ABB RAPID module: RsTempModule.mod

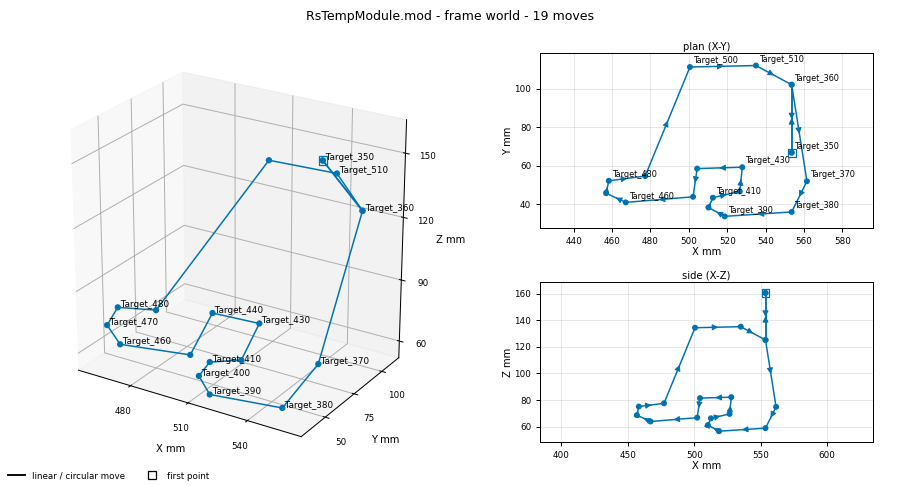
[picture p0: tool path of RsTempModule.mod in frame world, 19 of 19 moves have a stored position in this frame; points joined in program order, loops and branches not executed]
MODULE RsTempModule
    LOCAL CONST robtarget Target_350:=[[-145.225874554,122.068654602,-50.082052893],[0.707106781,0.000000819,-0.000000819,-0.707106781],[1,1,0,7],[9E+09,9E+09,9E+09,9E+09,9E+09,9E+09]];
    LOCAL PERS tooldata Portamarcador:=[TRUE,[[105.653,-1.591,36.465],[0.707106781,0,0.707106781,0]],[0.25,[0,0,1],[1,0,0,0],0,0,0]];
    LOCAL PERS wobjdata Tablero:=[FALSE,TRUE,"",[[0,0,0],[1,0,0,0]],[[431.492,204.933,227.769],[0.270598807,-0.653281169,-0.653281169,-0.270598807]]];
    LOCAL CONST robtarget Target_360:=[[-145.225990414,122.068654602,-0.082052893],[0.707106781,0.000000819,-0.000000819,-0.707106781],[0,0,0,1],[9E+09,9E+09,9E+09,9E+09,9E+09,9E+09]];
    LOCAL CONST robtarget Target_370:=[[-216.314272977,130.011265242,-0.08221762],[0.707106782,0.00000082,-0.000000819,-0.707106781],[-1,1,-2,0],[9E+09,9E+09,9E+09,9E+09,9E+09,9E+09]];
    LOCAL CONST robtarget Target_380:=[[-238.920712,122.070831135,-0.082270004],[0.707106781,0.00000082,-0.00000082,-0.707106781],[-1,1,-2,0],[9E+09,9E+09,9E+09,9E+09,9E+09,9E+09]];
    LOCAL CONST robtarget Target_390:=[[-242.176963668,87.21495429,-0.082277549],[0.707106781,0.000000819,-0.000000819,-0.707106781],[-1,1,-2,0],[9E+09,9E+09,9E+09,9E+09,9E+09,9E+09]];
    LOCAL CONST robtarget Target_400:=[[-235.683786475,78.752058887,-0.082262503],[0.707106781,0.000000819,-0.000000819,-0.707106781],[-1,1,-2,0],[9E+09,9E+09,9E+09,9E+09,9E+09,9E+09]];
    LOCAL CONST robtarget Target_410:=[[-228.457991082,81.055519424,-0.082245759],[0.707106781,0.000000819,-0.000000819,-0.707106781],[-1,1,-2,0],[9E+09,9E+09,9E+09,9E+09,9E+09,9E+09]];
    LOCAL CONST robtarget Target_420:=[[-223.813275477,95.060731266,-0.082234996],[0.707106781,0.000000819,-0.000000819,-0.707106781],[-1,1,-2,0],[9E+09,9E+09,9E+09,9E+09,9E+09,9E+09]];
    LOCAL CONST robtarget Target_430:=[[-205.993838978,96.347520237,-0.082193705],[0.707106781,0.000000819,-0.00000082,-0.707106781],[-1,1,-2,0],[9E+09,9E+09,9E+09,9E+09,9E+09,9E+09]];
    LOCAL CONST robtarget Target_440:=[[-207.00309405,72.842237427,-0.082196044],[0.707106782,0.000000819,-0.000000818,-0.707106781],[-1,1,-2,0],[9E+09,9E+09,9E+09,9E+09,9E+09,9E+09]];
    LOCAL CONST robtarget Target_450:=[[-227.772910705,70.716966245,-0.082244172],[0.707106781,0.000000819,-0.000000819,-0.707106781],[-1,1,-2,0],[9E+09,9E+09,9E+09,9E+09,9E+09,9E+09]];
    LOCAL CONST robtarget Target_460:=[[-231.882732587,35.693817055,-0.082253695],[0.707106781,0.000000819,-0.000000819,-0.707106781],[-1,1,-2,0],[9E+09,9E+09,9E+09,9E+09,9E+09,9E+09]];
    LOCAL CONST robtarget Target_470:=[[-225.128328942,25.434710387,-0.082238044],[0.707106781,0.000000819,-0.000000819,-0.707106781],[-1,1,-2,0],[9E+09,9E+09,9E+09,9E+09,9E+09,9E+09]];
    LOCAL CONST robtarget Target_480:=[[-215.976129925,26.869358271,-0.082216836],[0.707106781,0.00000082,-0.00000082,-0.707106781],[-1,1,-2,0],[9E+09,9E+09,9E+09,9E+09,9E+09,9E+09]];
    LOCAL CONST robtarget Target_490:=[[-212.521294514,45.774375392,-0.08220883],[0.707106781,0.000000819,-0.000000819,-0.707106781],[-1,1,-2,0],[9E+09,9E+09,9E+09,9E+09,9E+09,9E+09]];
    LOCAL CONST robtarget Target_500:=[[-132.204623558,69.10534384,-0.08202272],[0.707106781,0.000000819,-0.00000082,-0.707106781],[0,2,-2,0],[9E+09,9E+09,9E+09,9E+09,9E+09,9E+09]];
    LOCAL CONST robtarget Target_510:=[[-131.099190925,103.471454414,-0.082020159],[0.707106781,0.000000819,-0.000000819,-0.707106781],[0,2,-2,0],[9E+09,9E+09,9E+09,9E+09,9E+09,9E+09]];
    LOCAL CONST robtarget Target_520:=[[-145.225990414,122.068654602,-0.082052893],[0.707106781,0.000000819,-0.000000819,-0.707106781],[0,0,0,1],[9E+09,9E+09,9E+09,9E+09,9E+09,9E+09]];
    LOCAL CONST robtarget Target_530:=[[-145.225874554,122.068654602,-50.082052893],[0.707106781,0.000000819,-0.000000819,-0.707106781],[-1,1,-2,0],[9E+09,9E+09,9E+09,9E+09,9E+09,9E+09]];
PROC RsTempPath()
        MoveL Target_350,v30,z10,Portamarcador\WObj:=Tablero;
        MoveL Target_360,v30,z10,Portamarcador\WObj:=Tablero;
        MoveL Target_370,v30,z10,Portamarcador\WObj:=Tablero;
        MoveL Target_380,v30,z10,Portamarcador\WObj:=Tablero;
        MoveL Target_390,v30,z10,Portamarcador\WObj:=Tablero;
        MoveL Target_400,v30,z10,Portamarcador\WObj:=Tablero;
        MoveL Target_410,v30,z10,Portamarcador\WObj:=Tablero;
        MoveL Target_420,v30,z10,Portamarcador\WObj:=Tablero;
        MoveL Target_430,v30,z10,Portamarcador\WObj:=Tablero;
        MoveL Target_440,v30,z10,Portamarcador\WObj:=Tablero;
        MoveL Target_450,v30,z10,Portamarcador\WObj:=Tablero;
        MoveL Target_460,v30,z10,Portamarcador\WObj:=Tablero;
        MoveL Target_470,v30,z10,Portamarcador\WObj:=Tablero;
        MoveL Target_480,v30,z10,Portamarcador\WObj:=Tablero;
        MoveL Target_490,v30,z10,Portamarcador\WObj:=Tablero;
        MoveL Target_500,v30,z10,Portamarcador\WObj:=Tablero;
        MoveL Target_510,v30,z10,Portamarcador\WObj:=Tablero;
        MoveL Target_520,v30,z10,Portamarcador\WObj:=Tablero;
        MoveL Target_530,v30,z10,Portamarcador\WObj:=Tablero;
ENDPROC

ENDMODULE
